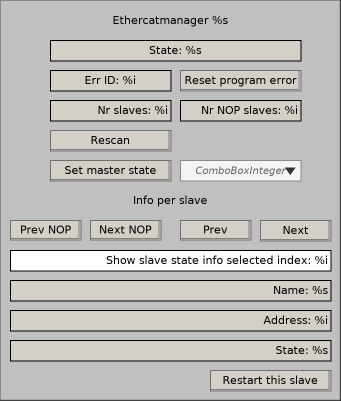
VISUALIZATION Vis_EthercatManager  // 341x401
VAR_IN_OUT
	IO_EM: cntrl_EthercatManager;
END_VAR
    Rectangle (0,0 341x401)
    Label (10,190 321x21), "Info per slave"
    Rectangle (50,100 121x21), "Nr slaves: %i", tooltip "Nr of found configured slaves", text variable: IO_EM.IO_STS.NrOfSlaves
    Button (180,220 71x20), "Prev"
        OnMouseDown: execute { IO_EM.IO_STS.IndexStatusCurrentDevice := IO_EM.IO_STS.IndexStatusCurrentDevice - 1; }
    Rectangle (10,10 321x21), "Ethercatmanager %s", text variable: IO_EM.fbEthercatDevicesManager.HM_AmsNetID
    Rectangle (10,250 321x21), "Show slave state info selected index: %i", text variable: IO_EM.IO_STS.IndexStatusCurrentDevice
        OnMouseClick: write the text variable via Default, min 0, max 100
    Button (260,220 71x21), "Next"
        OnMouseDown: execute { IO_EM.IO_STS.IndexStatusCurrentDevice := IO_EM.IO_STS.IndexStatusCurrentDevice + 1; }
    Rectangle (180,100 121x21), "Nr NOP slaves: %i", tooltip "Slaves not in "OP" state", text variable: IO_EM.IO_STS.NrOfSlavesNotInOp
    Rectangle (10,280 321x21), "Name: %s", tooltip "Slaves not in "OP" state", text variable: IO_EM.IO_STS.StatusSlaveDevice.Name
    Rectangle (10,310 321x21), "Address: %i", tooltip "Slaves not in "OP" state", text variable: IO_EM.IO_STS.StatusSlaveDevice.Address
    Rectangle (10,340 321x21), "State: %s", tooltip "Slaves not in "OP" state", text variable: IO_EM.IO_STS.StatusSlaveDevice.State
    Button (50,130 121x21), "Rescan", pressed state: IO_EM.IO_STS.PB_UpdateConfigAndStates
        toggle IO_EM.IO_STS.PB_UpdateConfigAndStates
    Button (50,160 121x21), "Set master state", pressed state: IO_EM.IO_STS.PB_SetMasterState
        toggle IO_EM.IO_STS.PB_SetMasterState
    Button (10,220 71x20), "Prev NOP"
        tap IO_EM.IO_STS.PB_JumpIndexToPreviousNotOpDevice
    Button (90,220 71x20), "Next NOP"
        tap IO_EM.IO_STS.PB_JumpIndexToNextNotOpDevice
    ComboBoxInteger (180,160 121x21), variable: IO_EM.IO_STS.ReqMasterState, text list: 'tlEthercatState'
    Button (210,370 121x21), "Restart this slave", pressed state: IO_EM.IO_STS.PB_RestartCurrentDevice
        toggle IO_EM.IO_STS.PB_RestartCurrentDevice
    Rectangle (50,40 251x21), "State: %s", text variable: IO_EM.fbEthercatDevicesManager.eS
    Button (180,70 121x21), "Reset program error", colour toggle: IO_EM.IO_STS.Error, pressed state: IO_EM.IO_STS.PB_ResetError
        toggle IO_EM.IO_STS.PB_ResetError
    Rectangle (50,70 121x21), "Err ID: %i", text variable: IO_EM.IO_STS.ErrorNr
END_VISUALIZATION

(* stored: Version 1.1.0.1, ProductVersion 3.1.4024.12
   Visu Vis_EthercatManager: Id {3d40bd71-7620-0fcb-21c5-8acde55a495b} *)
